INTERFACE I_InputSourceHistorical EXTENDS I_InputSource

METHOD HistoricalCtrl : BOOL
VAR_INPUT
	stCtrl: REFERENCE TO ST_HMI_InputSourceCtrl;
	stHistStreamInfo: REFERENCE TO ST_HMI_DataSourceHist;
	stRecordInfo: REFERENCE TO ST_HMI_DataSourceHistRecordInfo;
END_VAR
END_METHOD

METHOD UpdateRecordList : BOOL
VAR_INPUT
	sStreamSystemID: GUID;
	stHistStreamInfo: REFERENCE TO ST_HMI_DataSourceHist;
END_VAR
END_METHOD

PROPERTY bCtrlChanged : BOOL
GET
END_GET
END_PROPERTY

END_INTERFACE

(* stored: Itf I_InputSourceHistorical: Id 70da735d-50c2-4123-b575-97450fe218cb
   Method HistoricalCtrl: Id f394cded-78f4-45ef-8d17-feb2823c41a6
   Method UpdateRecordList: Id 033a7b17-9d97-4081-b3c3-187d4d446fa3
   Property bCtrlChanged: Id 63bdf16c-4ca3-40ad-92e2-8852802c1823
   Get Get: Id ebaef1b4-57b3-4e28-8c47-1dc006514ef5 *)
